TEXTLIST TextList_Config_Mouvements
  0 = '' | FR: 'Rotation' | EN: 'Rotation'
  1 = '' | FR: 'Tilt' | EN: 'Tilt'
  2 = '' | FR: "Décalage d'origine" | EN: 'Home shift'
  3 = '' | FR: 'Erreur max. de vitesse' | EN: 'Max. speed error'
  4 = '' | FR: 'Retard défaut de surveillance vitesse' | EN: 'Speed monitoring error delay'
  5 = '' | FR: 'Limitation de couple' | EN: 'Torque limitation'
   = ''
END_TEXTLIST

(* stored: Version 1.1.0.1, ProductVersion 3.1.4024.10
   TextList TextList_Config_Mouvements: Id {594afd67-e55a-4474-a429-828b7409599b} *)
